FUNCTION_BLOCK boolMerge (* Basic Function Block Type *)
  (* Standard: 61499-2 *)
  (* Version 0.0, 14/02/2014, Gulnar zhan, nxtControl GmbH, Template *)
  PACKAGE Main;
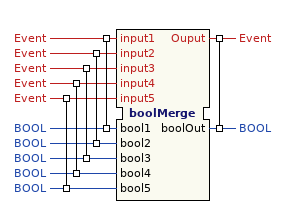
  EVENT_INPUT
    input1 WITH bool1;
    input2 WITH bool2;
    input3 WITH bool3;
    input4 WITH bool4;
    input5 WITH bool5;
  END_EVENT
  EVENT_OUTPUT
    Ouput WITH boolOut;
  END_EVENT
  VAR_INPUT
    bool1 : BOOL;
    bool2 : BOOL;
    bool3 : BOOL;
    bool4 : BOOL;
    bool5 : BOOL;
  END_VAR
  VAR_OUTPUT
    boolOut : BOOL;
  END_VAR
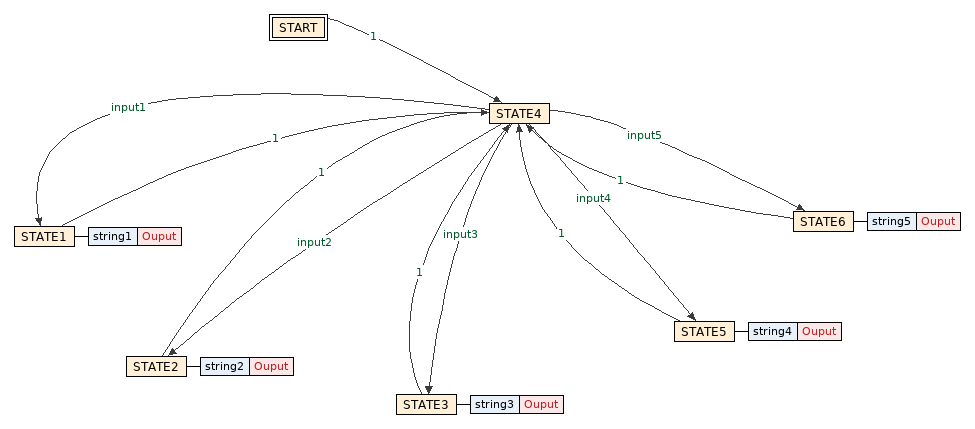
  EC_STATES
    START; (* Initial State *)
    STATE1 : string1 -> Ouput;
    STATE2 : string2 -> Ouput;
    STATE3 : string3 -> Ouput;
    STATE4;
    STATE5 : string4 -> Ouput;
    STATE6 : string5 -> Ouput;
  END_STATES
  EC_TRANSITIONS
    STATE4 TO STATE1 := input1;
    STATE4 TO STATE2 := input2;
    STATE4 TO STATE3 := input3;
    STATE1 TO STATE4 := 1;
    STATE2 TO STATE4 := 1;
    STATE3 TO STATE4 := 1;
    START TO STATE4 := 1;
    STATE4 TO STATE5 := input4;
    STATE5 TO STATE4 := 1;
    STATE4 TO STATE6 := input5;
    STATE6 TO STATE4 := 1;
  END_TRANSITIONS
  ALGORITHM string1 IN ST: (* Normally executed algorithm *)
;
(*stringOut:= '';*)
boolOut:= bool1;
  END_ALGORITHM
  ALGORITHM string2 IN ST:
;
(*stringOut:= '';*)
boolOut:= bool2;
  END_ALGORITHM
  ALGORITHM string3 IN ST:
;
(*stringOut:= '';*)
boolOut:= bool3;
  END_ALGORITHM
  ALGORITHM string4 IN ST:
;
boolOut:= bool4;
  END_ALGORITHM
  ALGORITHM string5 IN ST:
;
boolOut:= bool5;
  END_ALGORITHM
END_FUNCTION_BLOCK
